FUNCTION_BLOCK FutureMCSetPositionCreator IMPLEMENTS InterfaceTaskCreator
VAR_INPUT
END_VAR
VAR_OUTPUT
END_VAR
VAR
	_axis: REFERENCE TO AXIS_REF;
	_position	: MC_LREAL;
	_mode		: BOOL;
	_option 	: ST_SetPositionOptions;
	_error_id :UDINT;
END_VAR

{warning 'add method implementation '}
METHOD create_future : InterfaceFuture
VAR_INPUT
	(* Specify future name*)
	future_name	: STRING;
END_VAR
VAR
	_p_future : POINTER TO FutureMCSetPosition;
END_VAR
_p_future := __NEW(FutureMCSetPosition);
_p_future^.future_name := future_name;
_p_future^.set_parameters(_axis, _position);
_p_future^.set_options(_mode, _option);
create_future := _p_future^;
END_METHOD

{warning 'add method implementation '}
METHOD destroy_future : InterfaceFuture
VAR_INPUT
	(* Specify future instance whtat you want to delete.*)
	future	: InterfaceFuture;
END_VAR
VAR
	_p_future : POINTER TO FutureMCSetPosition;
END_VAR
IF __QUERYPOINTER(future, _p_future) THEN
	__DELETE(_p_future);
	IF _p_future = 0  THEN
		destroy_future := 0;
	END_IF
END_IF
END_METHOD

METHOD set_options : BOOL
VAR_INPUT
	mode		: BOOL;
	option 	: ST_SetPositionOptions;
END_VAR
_mode := mode;
_option := option;
END_METHOD

METHOD set_parameters : BOOL
VAR_INPUT
	axis: REFERENCE TO AXIS_REF;
	position	: MC_LREAL;
END_VAR
_axis REF= axis;
_position := position;
END_METHOD

END_FUNCTION_BLOCK

(* stored: Version 1.1.0.1, ProductVersion 3.1.4024.15
   POU FutureMCSetPositionCreator: Id {293e97ce-3a12-4515-9239-8cf3983d688e}, SpecialFunc None
   Method create_future: Id {0f731815-c09f-4a7d-a2aa-84ddc0096e42}
   Method destroy_future: Id {d7f6d590-731b-46b0-9c94-43523208ac96}
   Method set_options: Id {c9ebcb01-df3f-4a2f-bbb7-ab2453c9dd29}
   Method set_parameters: Id {30243bcd-4b24-4548-9612-359c1e0c45d0} *)
